Fanuc KAREL source: compact_preamble.KL

PROGRAM KT00082
%NOLOCKGROUP
VAR
Y1 : ARRAY[2] OF BYTE
I2:INTEGER
OUT:REAL
BEGIN
Y1[1]=2
I2=3
OUT=((Y1[1] * I2))
END KT00082
